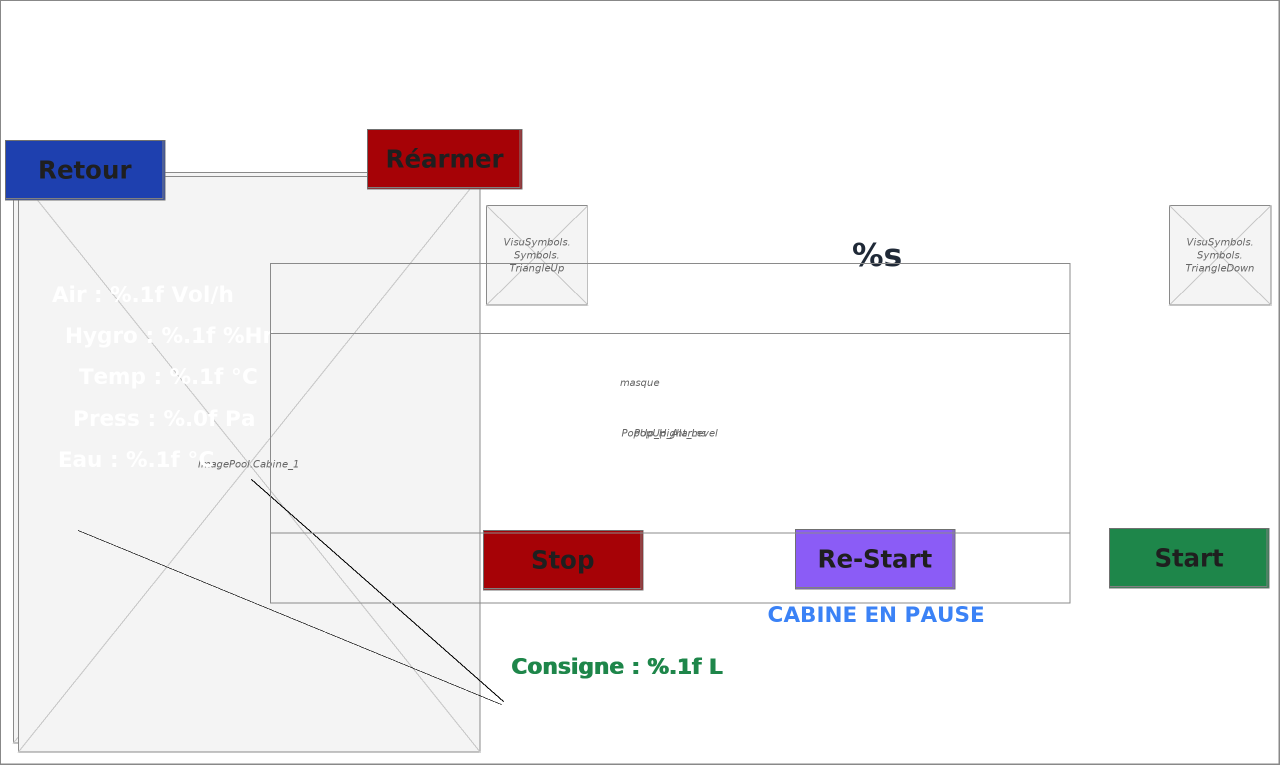
VISUALIZATION ModeManuel  // 1280x765
    Frame (0,0 1280x765)
        shows masque()
    Image (13,172 466x571), image: ImagePool.Cabine-2
    Polygon (40,654) (180,695) (321,730) (395,695) (469,654), colour variable: GVL_Visu.Couleur_Cabine
    Polygon (42,654) (40,249) (323,189) (466,256) (467,654), colour variable: GVL_Visu.Couleur_Cabine
    Image (18,176 462x576), image: ImagePool.Cabine_1
        OnMouseDown: OpenDialog Dialog=Actionneurs, OpenModal=True, OpenCentered=True
    Button (5,140 160x60), "Retour", invisible if: Mode_Cabine_Manuel
        OnMouseDown: change screen: menu
    Group (49,274 322x206)
        Rectangle (13,41 295x41), "Hygro : %.1f %Hr", text variable: Tab_MES_Sonde_Hygro_Amb.R_MesCor
        Rectangle (27,82 295x41), "Temp : %.1f °C", text variable: Tab_MES_Sonde_Temp_Amb.R_MesCor
        Rectangle (0,0 295x41), "Air : %.1f Vol/h", text variable: MES_Debit_Volh_Soufflage, invisible if: TRUE
        Rectangle (21,124 295x41), "Press : %.0f Pa", text variable: Tab_MES_Sonde_Press_Cab.R_MesCor
        Rectangle (6,165 295x41), "Eau : %.1f °C", text variable: MES_Temp_Eau_Mitige_General
    Rectangle (507,613 294x41), "Débit : %.1f l/min", text variable: GVL_Visu.Visu_Mes_Debit_Eau_Manu, invisible if: NOT GVL_Visu.Visu_Debit_Eau_Manu
    Group (486,205 100x100), invisible if: Mode_Cabine_Manuel
        OnMouseDown: execute {
            Manu_Choix_Numero_Mode := Manu_Choix_Numero_Mode - 1;
            IF (Manu_Choix_Numero_Mode < GVL_Visu.Min_Mode_Manu)
            	THEN
            	Manu_Choix_Numero_Mode := GVL_Visu.Min_Mode_Manu;
            END_IF
            GVL_Visu.Manu_i := 30;
            FOR GVL_Visu.Manu_i := 30 TO 0 BY -1 DO
            	IF ((NOT GVL_Visu.Tab_Choix_Modes[GVL_Visu.Manu_i]) AND (Manu_Choix_Numero_Mode = GVL_Visu.Manu_i))
            		THEN
            		Manu_Choix_Numero_Mode := Manu_Choix_Numero_Mode - 1;
            	END_IF
            END_FOR
        }
        Button (0,0 100x100)
        Image (0,0 102x100), image: VisuSymbols.Symbols.TriangleUp
    RoundedRectangle (588,205 579x100), "%s", text list: 'Noms_Modes', text index: GVL_Visu.Manu_Choix_Numero_Mode_INT
    Group (1169,205 100x100), invisible if: Mode_Cabine_Manuel
        OnMouseDown: execute {
            Manu_Choix_Numero_Mode := Manu_Choix_Numero_Mode + 1;
            GVL_Visu.Manu_j := 0;
            FOR GVL_Visu.Manu_j := 0 TO 29 BY 1 DO
            	IF (NOT (GVL_Visu.Tab_Choix_Modes[GVL_Visu.Manu_j]) AND (Manu_Choix_Numero_Mode = GVL_Visu.Manu_j))
            		THEN
            		Manu_Choix_Numero_Mode := Manu_Choix_Numero_Mode + 1;
            	END_IF
            END_FOR
            IF (Manu_Choix_Numero_Mode > GVL_Visu.Max_Mode_Manu)
            	THEN
            	Manu_Choix_Numero_Mode := GVL_Visu.Max_Mode_Manu;
            END_IF
        }
        Button (0,0 100x100)
        Image (0,0 102x100), image: VisuSymbols.Symbols.TriangleDown
    Button (367,129 155x60), "Réarmer", invisible if: NOT Condi_Affich_Rearm
        OnMouseDown: toggle Cmd_Rearmement
    Rectangle (588,170 186x41), "Mode N°%d", text variable: GVL_Visu.Manu_Choix_Numero_Mode_INT
    Button (1109,528 160x60), "Start", invisible if: Mode_Cabine_Manuel
        OnMouseDown: toggle Start_Mode_Manu
    Group (483,329 786x263), invisible if: Mode_Cabine_Manuel
        Group (445,67 341x63), invisible if: NOT GVL_Visu.Affich_Debit_Eau_Manu_Douche
            Rectangle (0,0 187x63), "Vol. d'eau :"
            RoundedRectangle (187,0 154x63), "%.1f L", text variable: Manu_Lct_Cons_Vol_Douche
                OnMouseDown: write the text variable via VisuDialogs.Numpad, min 0, max 100, format %0.1f
        Group (0,0 445x63), invisible if: GVL_Visu.Affich_Debit_Eau_Manu
            Rectangle (0,0 186x63), "Heure(s) :"
            RoundedRectangle (186,0 259x63), "%.0f heure(s)", text variable: Manu_Tempo_Transition_Heure
                OnMouseDown: write the text variable via VisuDialogs.Numpad, min 0, max 23, format %.0f
        Group (0,67 445x63), invisible if: GVL_Visu.Affich_Debit_Eau_Manu
            Rectangle (0,0 186x63), "Minute(s) :"
            RoundedRectangle (186,0 259x63), "%.0f minute(s)", text variable: Manu_Tempo_Transition_Minute
                OnMouseDown: write the text variable via VisuDialogs.Numpad, min 0, max 59, format %.0f
        Group (0,133 445x63), invisible if: GVL_Visu.Affich_Debit_Eau_Manu
            Rectangle (0,0 186x63), "Seconde(s) :"
            RoundedRectangle (186,0 259x63), "%.0f seconde(s)", text variable: Manu_Tempo_Transition_Seconde
                OnMouseDown: write the text variable via VisuDialogs.Numpad, min 0, max 59, format %.0f
        Group (445,0 341x63), invisible if: GVL_Visu.Manu_Choix_Numero_Mode_INT = 8
            Rectangle (0,0 187x63), "Ventilation :"
            RoundedRectangle (187,0 154x63), "%.0f Vol/h", text variable: Manu_Cons_Deb_Soufflage
                OnMouseDown: write the text variable via VisuDialogs.Numpad, min 0, max 200, format %.0f
        Group (0,200 445x63), invisible if: NOT GVL_Visu.Affich_ChasseEau_Manu
            Rectangle (0,0 186x63), "Nbre chasse :"
            RoundedRectangle (186,0 259x63), "%.0f", text variable: Manu_Cons_Nbre_Chasse
                OnMouseDown: write the text variable via VisuDialogs.Numpad, min 0, max 99, format %.0f
        Group (445,133 341x63), invisible if: NOT GVL_Visu.Visu_Temp_Manu
            Rectangle (0,0 187x63), "Temp. eau :"
            RoundedRectangle (187,0 154x63), "%.0f °C", text variable: Manu_Cons_Temp_Eau
                OnMouseDown: write the text variable via VisuDialogs.Numpad, min 10, max 50, format %.0f
        Group (445,67 341x63), invisible if: NOT GVL_Visu.Affich_Debit_Eau_Manu_Lavabo
            Rectangle (0,0 187x63), "Vol. d'eau :"
            RoundedRectangle (187,0 154x63), "%.1f L", text variable: Manu_Lct_Cons_Vol_Lavabo
                OnMouseDown: write the text variable via VisuDialogs.Numpad, min 0, max 100, format %0.1f
    Group (483,129 650x506), invisible if: NOT Mode_Cabine_Manuel
        Button (312,400 160x60), "Pause", invisible if: Statut_Pause_Force
            OnMouseDown: toggle Bp_Pause
        Rectangle (140,0 510x50), "MODE MANUEL EN COURS", invisible if: GVL_Visu.On_Off_Anim
        Button (0,401 160x60), "Stop"
            OnMouseDown: toggle Reset_Mode_Manu
        Button (312,400 160x60), "Re-Start", invisible if: NOT Statut_Pause_Force
            OnMouseDown: toggle Bp_Pause
        Group (172,208 446x165), invisible if: GVL_Visu.Affich_Debit_Eau_Manu
            Rectangle (11,0 322x41), "Heure(s) restante(s) :"
            Rectangle (333,0 113x41), "%.0f hrs", text variable: Temp_Restant_Heure
            Rectangle (11,83 322x41), "Seconde(s) restante(s) :"
            Rectangle (333,83 113x41), "%.0f sec", text variable: Temp_Restant_Seconde
            Rectangle (11,41 322x41), "Minute(s) restante(s) :"
            Rectangle (333,41 113x41), "%.0f min", text variable: Temp_Restant_Minute
            Group (0,124 446x41), invisible if: NOT GVL_Visu.Visu_ChasseEau_Manu
                Rectangle (0,0 322x41), "Chasse(s) restante(s) :"
                Rectangle (322,0 74x41), "%.0f /", text variable: Nbre_Chasse_EnCours
                Rectangle (388,0 58x41), "%.0f", text variable: Nbre_Chasse_Total
        Rectangle (246,465 294x41), "CABINE EN PAUSE", invisible if: GVL_Visu.On_Off_Anim OR NOT Comande_Pause
    Group (251,479 602x246), invisible if: NOT GVL_Visu.Visu_VolEau_Douche_Manu
        Line (0,0) (252,222)
        Rectangle (258,205 344x41), "Volume d'eau : %.1f L", text variable: Lect_Volume_Eau_Douche
        Rectangle (258,171 344x33), "Consigne : %.1f L", text variable: Manu_Lct_Cons_Vol_Douche
    Group (78,530 774x195), invisible if: NOT GVL_Visu.Visu_VolEau_Lavabo_Manu
        Line (0,0) (423,174)
        Rectangle (430,154 344x41), "Volume d'eau : %.1f L", text variable: Lect_Volume_Eau_Lavabo
        Rectangle (430,120 344x33), "Consigne : %.1f L", text variable: Manu_Lct_Cons_Vol_Lavabo
    Group (270,263 800x340)
        Frame (0,0 800x340), invisible if: NOT GVL_Visu.Affichage_PopUp_Alarm
            shows PopUp_Alarms()
        Frame (0,70 800x200), invisible if: NOT GVL_Visu.Affichage_PopUp_HightLevel
            shows PopUp_Hight_Level()
END_VISUALIZATION

(* stored: Version 1.1.0.1, ProductVersion 3.1.4024.16
   Visu ModeManuel: Id {df7010ee-0092-4eb0-9878-bae23da34b74} *)
